# EPICS IOC start-up script: iocsh/ethercatmcIndexerAxis.iocsh
ethercatmcCreateIndexerAxis("$(MOTOR_PORT)", "$(AXIS_NO)", "6", "$(AXISCONFIG)")

dbLoadRecords("ethercatmc.template", "P=$(P), R=$(R), MOTOR_PORT=$(MOTOR_PORT), ASYN_PORT=$(ASYN_PORT), AXIS_NO=$(AXIS_NO), PREC=$(PREC), HLSV=$(HLSV=0), RAWENCSTEP_ADEL=$(RAWENCSTEP_ADEL), RAWENCSTEP_MDEL=$(RAWENCSTEP_MDEL) $(ECAXISFIELDINIT)")

dbLoadRecords("ethercatmcAuxBitsStatus.template", "P=$(P), R=$(R), AXIS_NO=$(AXIS_NO), MOTOR_PORT=$(MOTOR_PORT), ASYN_PORT=$(ASYN_PORT), AXIS_NO=$(AXIS_NO) ")

dbLoadRecords("ethercatmcindexer.template", "P=$(P), R=$(R), MOTOR_PORT=$(MOTOR_PORT), ASYN_PORT=$(ASYN_PORT), AXIS_NO=$(AXIS_NO), PREC=$(PREC) ")

dbLoadRecords("ethercatmcreadback.template", "P=$(P), R=$(R), MOTOR_PORT=$(MOTOR_PORT), ASYN_PORT=$(ASYN_PORT), AXIS_NO=$(AXIS_NO), PREC=$(PREC), ALWAYS_GET_VELO=$(ALWAYS_GET_VELO=1)")
